(* Schneider Machine Expert - Basic project Zımpara-DIGITALINOUT, file version 1.8.0.0 *)
(* ProjectInformations: Name=Yeni proje *)

HARDWARE
  Cpu 0: TM221ME16T/G
  ModuleExtensionObject 0: TM3DI8/G
  ModuleExtensionObject 1: TM3AQ2/G
  EthernetConfiguration: NetworkName=M221, IpAllocationMode=FixedAddress, IpAddress=192.168.0.15, SubnetMask=255.255.255.0
  SerialLineConfiguration: Baud=Baud19200, Parity=ParityNone, DataBits=DataBits8, StopBits=StopBits1, PhysicalMedium=PhysicalMediumRs485, TransmissionMode=TransmissionModeModbusRtu, SlaveId=1, Addressing=SlaveAddressing
  MastTask: UsePeriodScanMode=false, PeriodScan=100
  FastTask: Period=255
  CpuBehavior: StartingMode=StartAsPreviousState, AutoSaveRamOnEeprom=true, WatchdogPeriod=250

SYMBOLS  (address, symbol, comment, settings)
  %M0         "HMI/OSILASYON YUKARI"
  %M1         "HMI/OSILASYON AŞAĞI"
  %M2         "HMI/FIRÇA  YUKARI"
  %M3         "HMI/FIRÇA  AŞAĞI"
  %M4         "HMI BANT START"
  %M5         "HMI OSILASYON START"
  %M6         "427/FIRCA INVERTOR"
  %M7         "428/VALF"
  %M8         "STOP"
  %M9         "HAFIZADAN ENCODERLERI ÇEK"
  %M10        "ENC 1 PRESET/OSILASYON ENC"
  %M11        "ENC 2 PRESET/FIRÇA ENC"
  %M12        "ENC_1_SIFIRLAMA/OSILASYON ENC"
  %M13        "ENC_2_SIFIRLAMA/FIRÇA ENC"
  %M16        "ENCODER2 ÇIKIŞ1"
  %M17        "ENCODER2 ÇIKIŞ2"
  %M18        "ENCODER2 ÇIKIŞ3"
  %M19        "ENCODER2 ÇIKIŞ4"
  %M21        "ENCODER 2 ÇIKIŞ1"
  %M22        "ENCODER 2 ÇIKIŞ2"
  %M23        "ENCODER 2 ÇIKIŞ3"
  %M24        "ENCODER 2 ÇIKIŞ4"
  %M26        "OSILASYON YÜKSEKLİK AYAR"
  %M27        "OSİLASYON YUKARI SET"
  %M28        "OSİLASYON AŞAĞI SET"
  %M29        "FIRÇA_YÜKSEKLİK_AYAR"
  %M30        "FIRÇA_YUKARI_SET"
  %M31        "FIRÇA_AŞAĞI_SET"
  %M32        "SQ5 CEVAP1"
  %M33        "SQ5 CEVAP2"
  %M201       "OSILASYON_KALIBRASYON"
  %S93      SB_MWBACKUP  "User set this bit to 1 to store the %MW variable in the flash (up to 2000)"
  %S94      SB_MWRESTORE  "User set this bit to 1 to restore the saved data"
  %SW148    SW_NBPERS  "Number of persistent variables (maximum 2000)"
  %MW1        "ENCODER 1 ÖN AYAR"
  %MW2        "ENCODER 2 ÖN AYAR"
  %MW30       "OSİLASYON SÜRÜCÜSÜ ANALOG ÇIKIŞ"
  %MW34       "ARKA FIRÇA SÜRÜCÜSÜ ANALOG ÇIKIŞ"
  %MW50       "BİRİNCİ ENKODER ANLIK DEĞERİ"
  %MW52       "İKİNCİ ENKODER ANLIK  DEĞERİ"
  %MF21       "2.ENCODER FLOAT DEĞERİ(MM)"
  %MF23       "1.ENKODER FLOAT DEĞERİ(MM)"
  %MF60       "ENC 1 FLOAT"
  %MF64       "OSILASYON MM YUKSEKLIK"
  %MF68       "OSILASYON ISTENEN YUKSEKLIK"
  %MF72       "ENC 2 FLOAT DEĞER"
  %MF76       "FIRÇA MM YÜKSEKLIK"
  %MF80       "FIRÇA ISTENEN YÜKSEKLIK"
  %MF84       "ENCODER 1 ÖN AYAR MM"
  %MF88       "ENCODER 1 ÖN AYAR INTEGER"
  %C0         "HAFIZADAN ENKODERLERİ ÇEK"
  %R0         "ENKODER 1 HAFIZAYA AT"
  %R1         "ENKODER 2 HAFIZAYA AT"
  %I0.0       "403/FIRÇA1 ÜST SINIR ANAHTARI"
  %I0.1       "402/FIRÇA1 ALT SINIR ANAHTARI"
  %I0.2       "405/FIRÇA2/ÜST SINIR ANAHTARI"
  %I0.3       "404/FIRÇA2/ ALT SINIR ANAHTARI"
  %I0.4       "SQ5(ÖN ARKA MESAFE SWITCHI)"
  %Q0.0       "421/OSİLASYON YUKARI"
  %Q0.1       "422/OSİLASYON AŞAĞI"
  %Q0.2       "423/FIRÇA 2 YUKARI"
  %Q0.3       "424/FIRÇA 2 AŞAĞI"
  %Q0.4       "425/BANT START"
  %Q0.5       "426/OSILASYON START"
  %Q0.6       "427/FIRCA INVERTER"
  %Q0.7       "428/VALF"
  %HSC0       "FIRÇA1/ENKODER"  [Type=CounterOrDownCounterBiPhasesX1, Preset=0, DedicatedInputs(DedicatedInput(Activated=true), DedicatedInput(Activated=true)), ReflexOutputs(ReflexOutput(Activated=false, LessThanS0=false, GreaterOrEqualThanS0=false, GreaterOrEqualThanS1=false), ReflexOutput(Activated=false, LessThanS0=false, GreaterOrEqualThanS0=false, GreaterOrEqualThanS1=false)), Thresholds(Threshold(ThresholdType=NotUsed, Pri]
  %HSC1       "FIRÇA2/ENKODER"  [Type=CounterOrDownCounterBiPhasesX1, Preset=0, DedicatedInputs(DedicatedInput(Activated=true), DedicatedInput(Activated=true)), ReflexOutputs(ReflexOutput(Activated=false, LessThanS0=false, GreaterOrEqualThanS0=false, GreaterOrEqualThanS1=false), ReflexOutput(Activated=false, LessThanS0=false, GreaterOrEqualThanS0=false, GreaterOrEqualThanS1=false)), Thresholds(Threshold(ThresholdType=NotUsed, Pri]
  %I1.0       "403/FIRÇA UST SINIR SWITCH"
  %I1.1       "402/FIRÇA ALT SINIR SWITCH"
  %I1.2       "405/FIRÇA2/ÜST SINIR SWITCH"
  %I1.3       "404/FIRÇA2/ALT SINIR SWITCH"
  %QW2.0      [Type=Type_0_10V, Scope=Scope_Customized, Minimum=0, Maximum=100]
  %QW2.1      [Type=Type_0_10V, Scope=Scope_Customized, Minimum=0, Maximum=100]

POU Yeni POU
  (* SectionNumber=1 *)

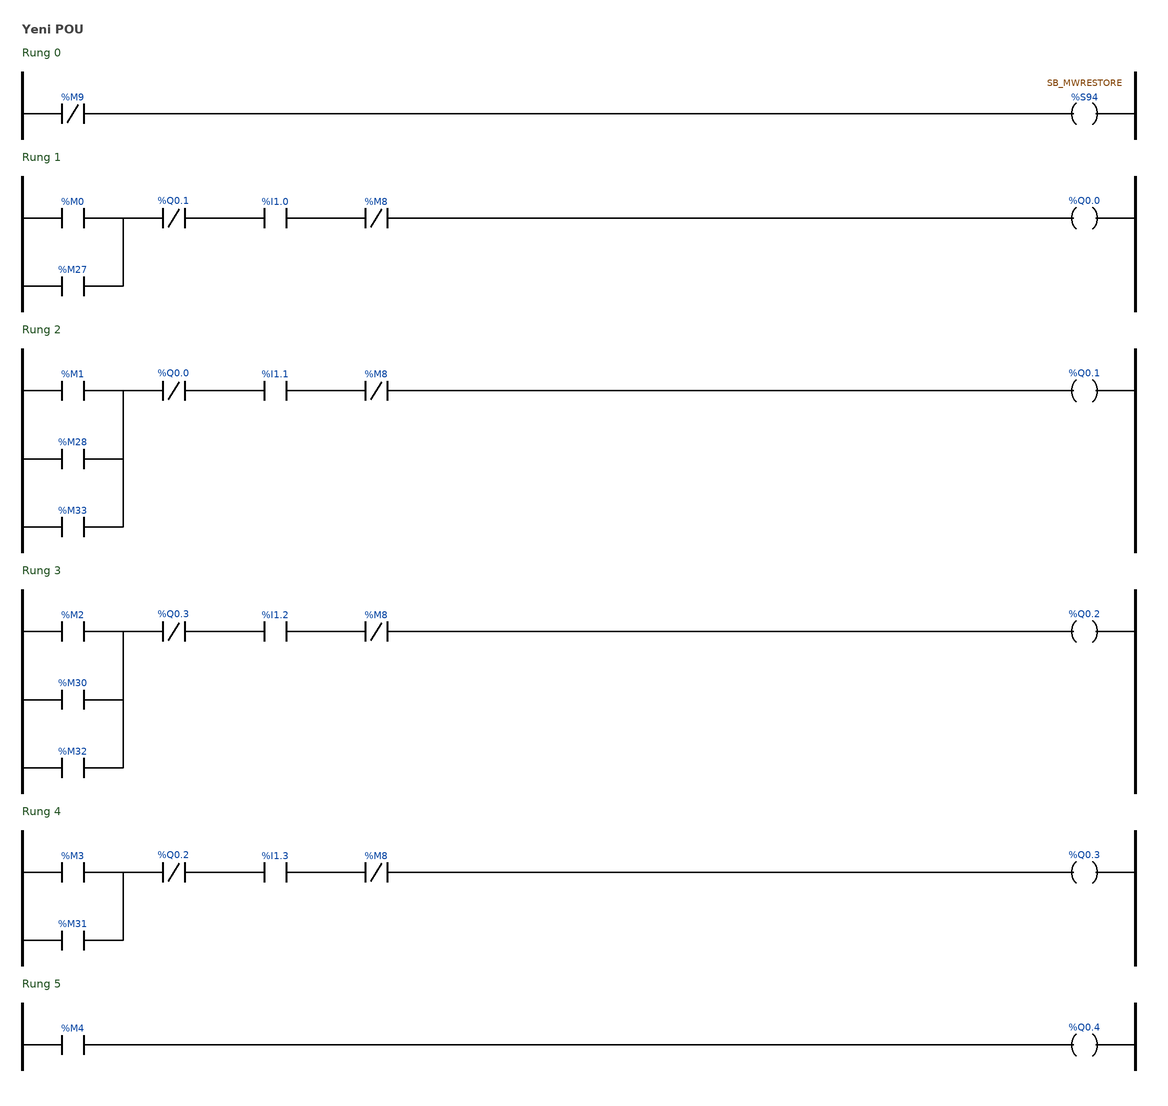

// Rung 0
  LDN %M9
  ST %S94                 (* SB_MWRESTORE *)
  // as ST:
  //   SB_MWRESTORE := NOT %M9;

// Rung 1
  LD %M0
  OR %M27
  ANDN %Q0.1
  AND %I1.0
  ANDN %M8
  ST %Q0.0
  // as ST:
  //   %Q0.0 := (%M0 OR %M27) AND NOT %Q0.1 AND %I1.0 AND NOT %M8;

// Rung 2
  LD %M1
  OR %M28
  OR %M33
  ANDN %Q0.0
  AND %I1.1
  ANDN %M8
  ST %Q0.1
  // as ST:
  //   %Q0.1 := (%M1 OR %M28 OR %M33) AND NOT %Q0.0 AND %I1.1 AND NOT %M8;

// Rung 3
  LD %M2
  OR %M30
  OR %M32
  ANDN %Q0.3
  AND %I1.2
  ANDN %M8
  ST %Q0.2
  // as ST:
  //   %Q0.2 := (%M2 OR %M30 OR %M32) AND NOT %Q0.3 AND %I1.2 AND NOT %M8;

// Rung 4
  LD %M3
  OR %M31
  ANDN %Q0.2
  AND %I1.3
  ANDN %M8
  ST %Q0.3
  // as ST:
  //   %Q0.3 := (%M3 OR %M31) AND NOT %Q0.2 AND %I1.3 AND NOT %M8;

// Rung 5
  LD %M4
  ST %Q0.4
  // as ST:
  //   %Q0.4 := %M4;

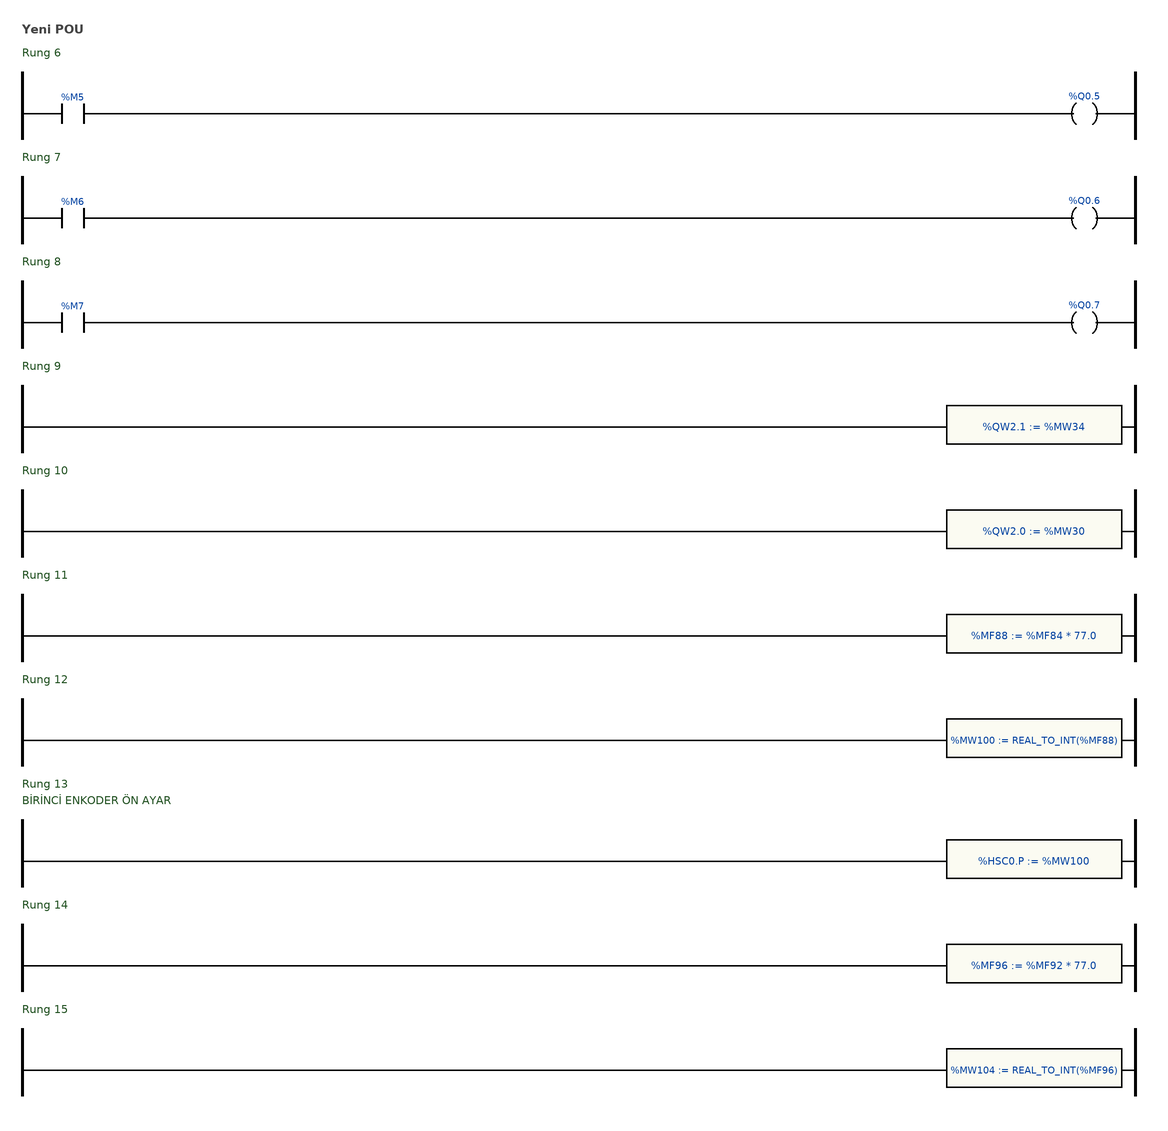

// Rung 6
  LD %M5
  ST %Q0.5
  // as ST:
  //   %Q0.5 := %M5;

// Rung 7
  LD %M6
  ST %Q0.6
  // as ST:
  //   %Q0.6 := %M6;

// Rung 8
  LD %M7
  ST %Q0.7
  // as ST:
  //   %Q0.7 := %M7;

// Rung 9
  LD 1
  [ %QW2.1 := %MW34 ]
  // as ST:
  //   %QW2.1 := %MW34;

// Rung 10
  LD 1
  [ %QW2.0 := %MW30 ]
  // as ST:
  //   %QW2.0 := %MW30;

// Rung 11
  LD 1
  [ %MF88 := %MF84 * 77.0 ]
  // as ST:
  //   %MF88 := %MF84  *  77.0;

// Rung 12
  LD 1
  [ %MW100 := REAL_TO_INT ( %MF88 ) ]
  // as ST:
  //   %MW100 := REAL_TO_INT ( %MF88 );

// Rung 13
// BİRİNCİ ENKODER ÖN AYAR
  LD 1
  [ %HSC0.P := %MW100 ]
  // as ST:
  //   %HSC0.P := %MW100;

// Rung 14
  LD 1
  [ %MF96 := %MF92 * 77.0 ]
  // as ST:
  //   %MF96 := %MF92  *  77.0;

// Rung 15
  LD 1
  [ %MW104 := REAL_TO_INT ( %MF96 ) ]
  // as ST:
  //   %MW104 := REAL_TO_INT ( %MF96 );

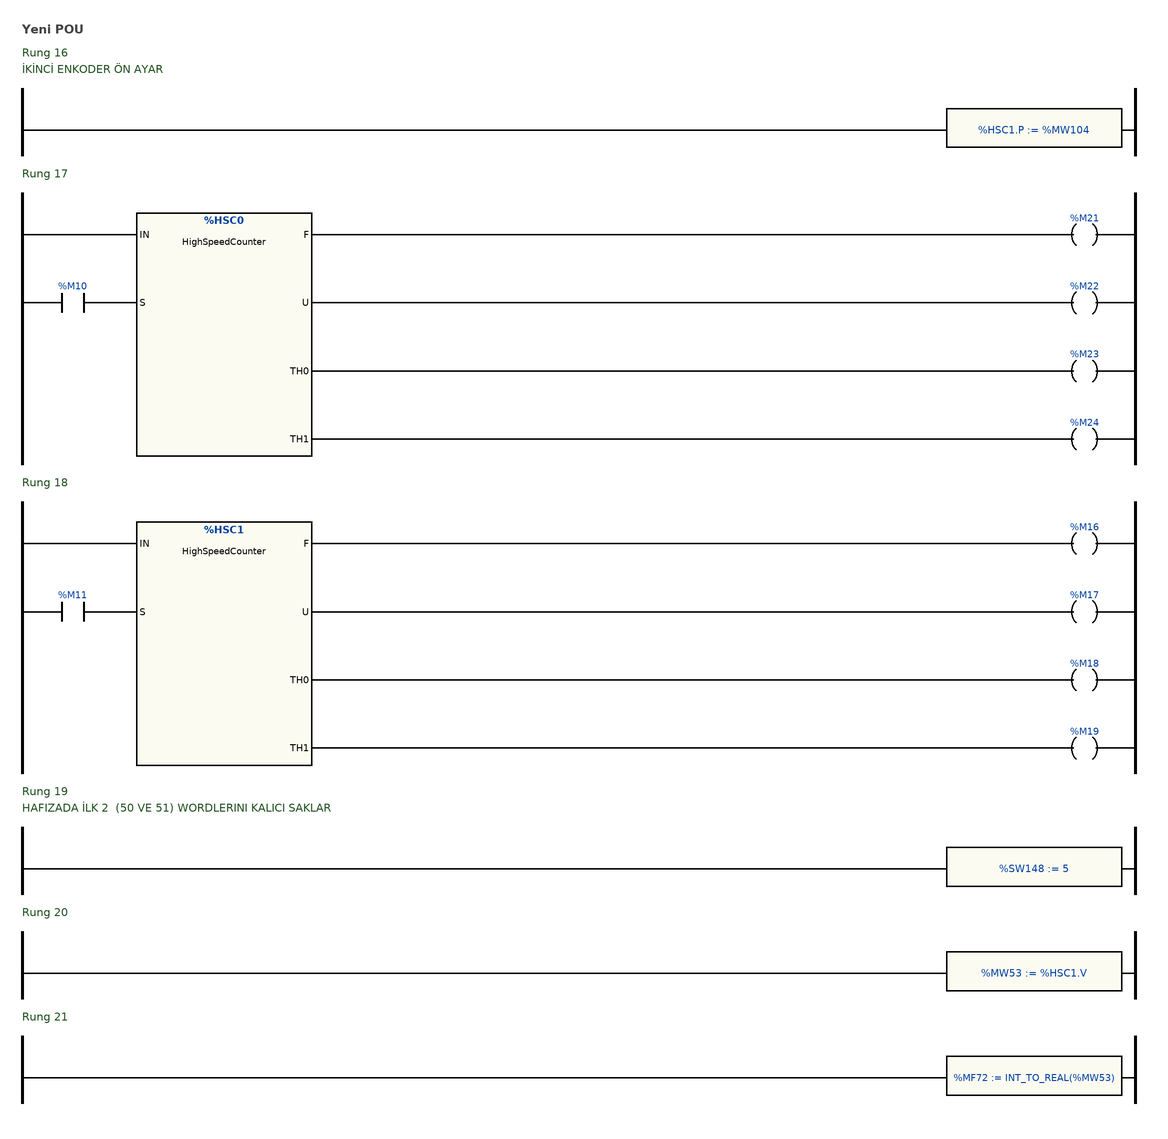

// Rung 16
// İKİNCİ ENKODER ÖN AYAR
  LD 1
  [ %HSC1.P := %MW104 ]
  // as ST:
  //   %HSC1.P := %MW104;

// Rung 17
  BLK %HSC0
  LD 1
  IN
  LD %M10
  S
  OUT_BLK
  LD F
  ST %M21
  LD U
  ST %M22
  LD TH0
  ST %M23
  LD TH1
  ST %M24
  END_BLK
  // as ST:
  //   %HSC0(IN := TRUE, S := %M10);
  //   %M21 := %HSC0.F;
  //   %M22 := %HSC0.U;
  //   %M23 := %HSC0.TH0;
  //   %M24 := %HSC0.TH1;

// Rung 18
  BLK %HSC1
  LD 1
  IN
  LD %M11
  S
  OUT_BLK
  LD F
  ST %M16
  LD U
  ST %M17
  LD TH0
  ST %M18
  LD TH1
  ST %M19
  END_BLK
  // as ST:
  //   %HSC1(IN := TRUE, S := %M11);
  //   %M16 := %HSC1.F;
  //   %M17 := %HSC1.U;
  //   %M18 := %HSC1.TH0;
  //   %M19 := %HSC1.TH1;

// Rung 19
// HAFIZADA İLK 2  (50 VE 51) WORDLERINI KALICI SAKLAR
  LD 1
  [ %SW148 := 5 ]         (* SW_NBPERS *)
  // as ST:
  //   SW_NBPERS := 5;

// Rung 20
  LD 1
  [ %MW53 := %HSC1.V ]
  // as ST:
  //   %MW53 := %HSC1.V;

// Rung 21
  LD 1
  [ %MF72 := INT_TO_REAL ( %MW53 ) ]
  // as ST:
  //   %MF72 := INT_TO_REAL ( %MW53 );

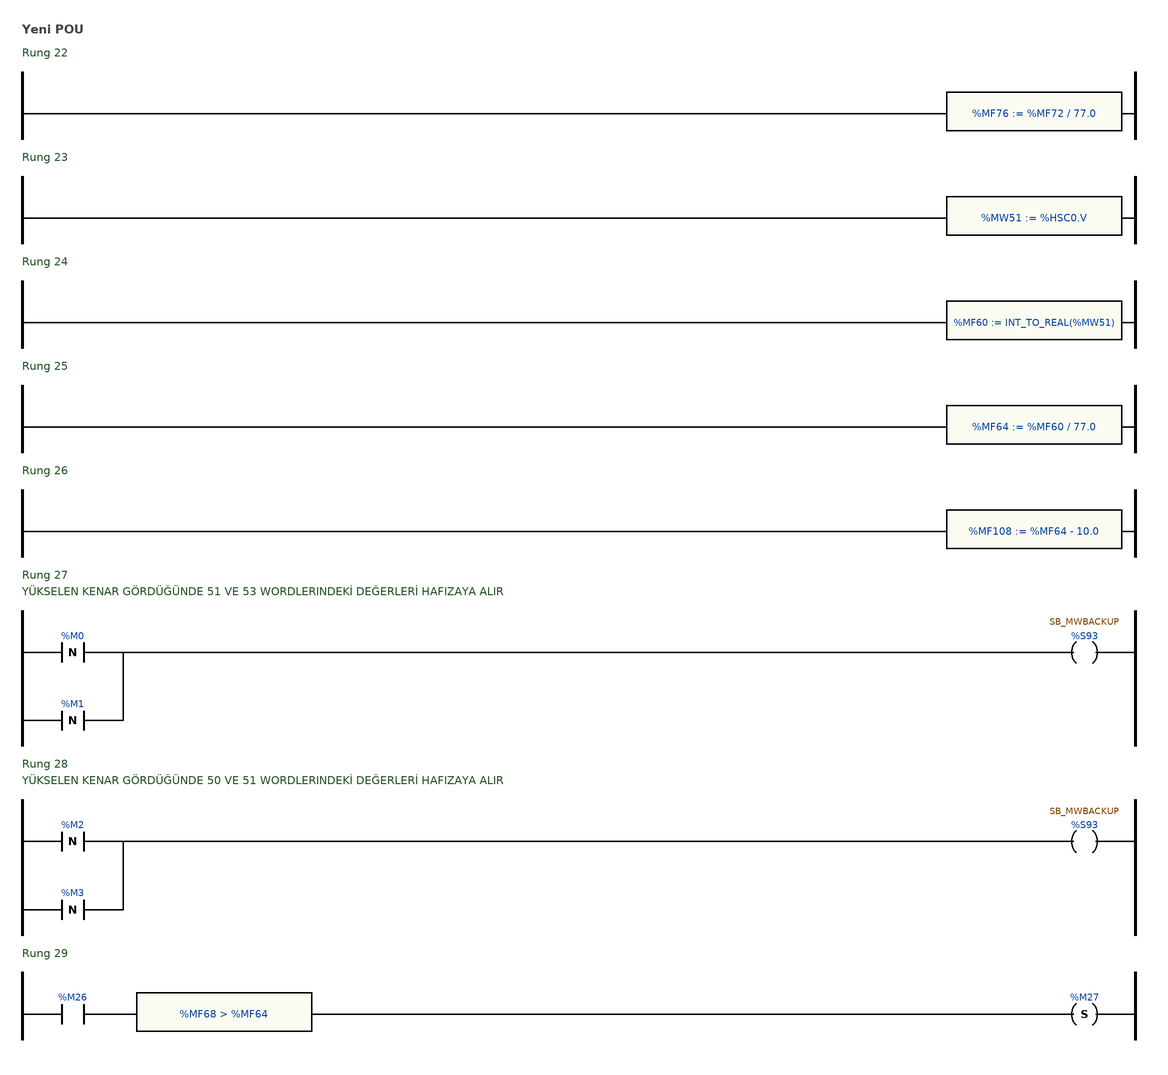

// Rung 22
  LD 1
  [ %MF76 := %MF72 / 77.0 ]
  // as ST:
  //   %MF76 := %MF72  /  77.0;

// Rung 23
  LD 1
  [ %MW51 := %HSC0.V ]
  // as ST:
  //   %MW51 := %HSC0.V;

// Rung 24
  LD 1
  [ %MF60 := INT_TO_REAL ( %MW51 ) ]
  // as ST:
  //   %MF60 := INT_TO_REAL ( %MW51 );

// Rung 25
  LD 1
  [ %MF64 := %MF60 / 77.0 ]
  // as ST:
  //   %MF64 := %MF60  /  77.0;

// Rung 26
  LD 1
  [ %MF108 := %MF64 - 10.0 ]
  // as ST:
  //   %MF108 := %MF64  -  10.0;

// Rung 27
// YÜKSELEN KENAR GÖRDÜĞÜNDE 51 VE 53 WORDLERINDEKİ DEĞERLERİ HAFIZAYA ALIR
  LDF %M0
  ORF %M1
  ST %S93                 (* SB_MWBACKUP *)
  // as ST:
  //   SB_MWBACKUP := FALLING(%M0) OR FALLING(%M1);

// Rung 28
// YÜKSELEN KENAR GÖRDÜĞÜNDE 50 VE 51 WORDLERINDEKİ DEĞERLERİ HAFIZAYA ALIR
  LDF %M2
  ORF %M3
  ST %S93                 (* SB_MWBACKUP *)
  // as ST:
  //   SB_MWBACKUP := FALLING(%M2) OR FALLING(%M3);

// Rung 29
  LD %M26
  AND [ %MF68 > %MF64 ]
  S %M27
  // as ST:
  //   IF %M26 AND %MF68 > %MF64 THEN %M27 := TRUE; END_IF;

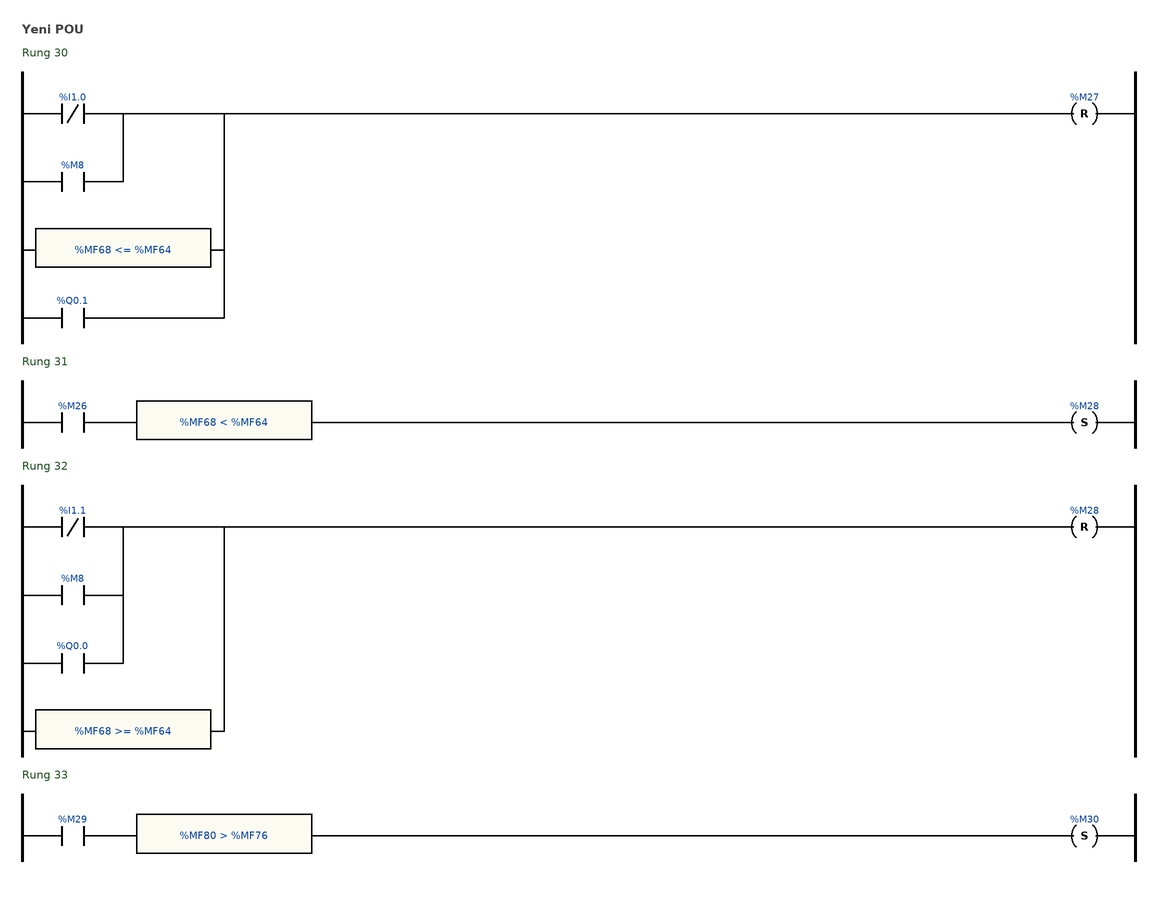

// Rung 30
  LDN %I1.0
  OR %M8
  OR [ %MF68 <= %MF64 ]
  OR %Q0.1
  R %M27
  // as ST:
  //   IF NOT %I1.0 OR %M8 OR %MF68 <= %MF64 OR %Q0.1 THEN %M27 := FALSE; END_IF;

// Rung 31
  LD %M26
  AND [ %MF68 < %MF64 ]
  S %M28
  // as ST:
  //   IF %M26 AND %MF68 < %MF64 THEN %M28 := TRUE; END_IF;

// Rung 32
  LDN %I1.1
  OR %M8
  OR %Q0.0
  OR [ %MF68 >= %MF64 ]
  R %M28
  // as ST:
  //   IF NOT %I1.1 OR %M8 OR %Q0.0 OR %MF68 >= %MF64 THEN %M28 := FALSE; END_IF;

// Rung 33
  LD %M29
  AND [ %MF80 > %MF76 ]
  S %M30
  // as ST:
  //   IF %M29 AND %MF80 > %MF76 THEN %M30 := TRUE; END_IF;

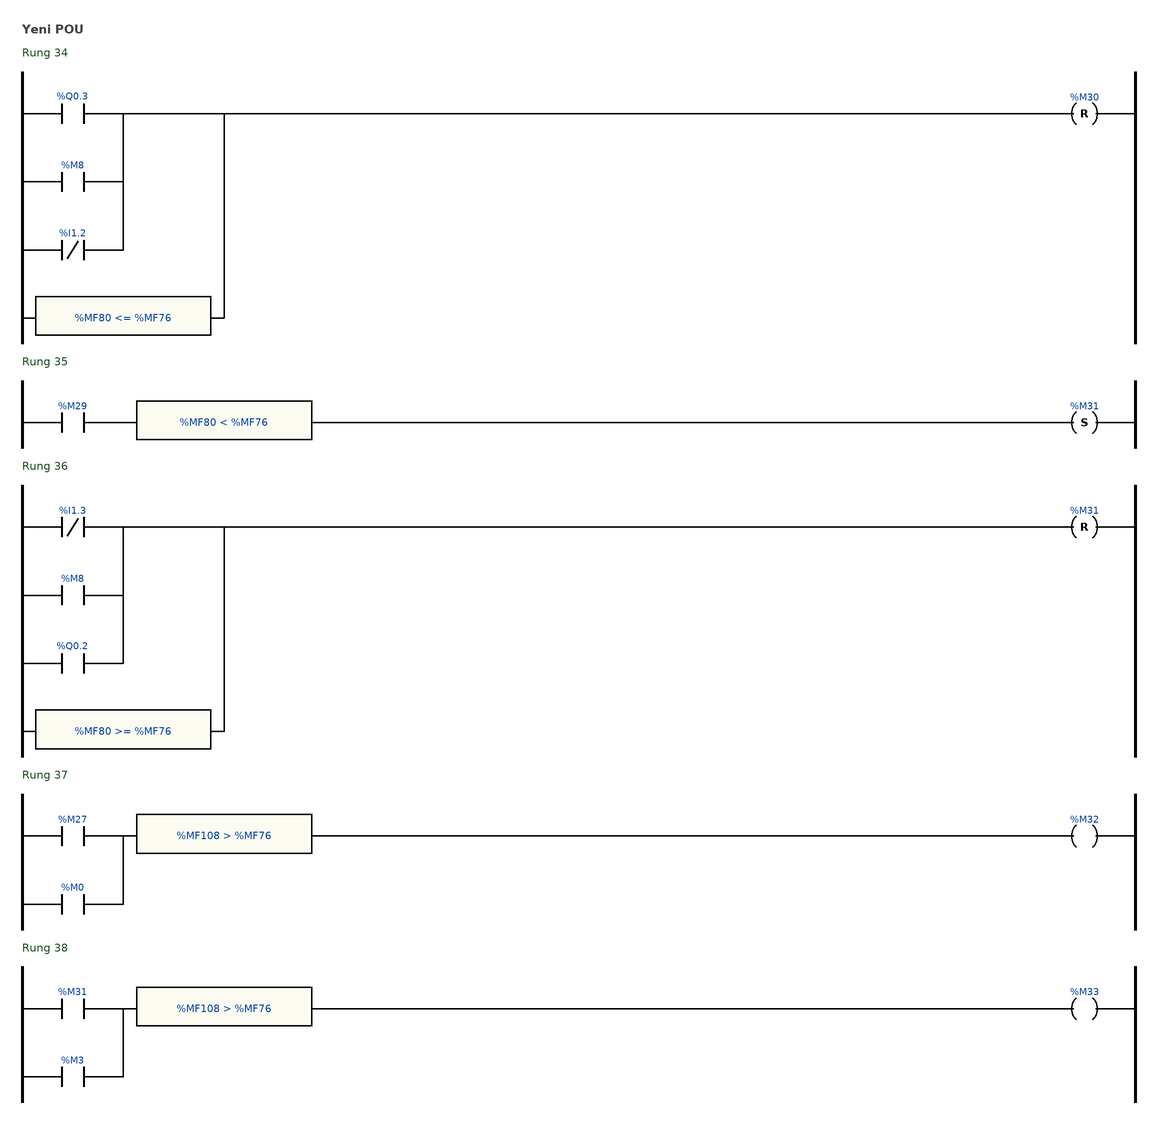

// Rung 34
  LD %Q0.3
  OR %M8
  ORN %I1.2
  OR [ %MF80 <= %MF76 ]
  R %M30
  // as ST:
  //   IF %Q0.3 OR %M8 OR NOT %I1.2 OR %MF80 <= %MF76 THEN %M30 := FALSE; END_IF;

// Rung 35
  LD %M29
  AND [ %MF80 < %MF76 ]
  S %M31
  // as ST:
  //   IF %M29 AND %MF80 < %MF76 THEN %M31 := TRUE; END_IF;

// Rung 36
  LDN %I1.3
  OR %M8
  OR %Q0.2
  OR [ %MF80 >= %MF76 ]
  R %M31
  // as ST:
  //   IF NOT %I1.3 OR %M8 OR %Q0.2 OR %MF80 >= %MF76 THEN %M31 := FALSE; END_IF;

// Rung 37
  LD %M27
  OR %M0
  AND [ %MF108 > %MF76 ]
  ST %M32
  // as ST:
  //   %M32 := (%M27 OR %M0) AND %MF108 > %MF76;

// Rung 38
  LD %M31
  OR %M3
  AND [ %MF108 > %MF76 ]
  ST %M33
  // as ST:
  //   %M33 := (%M31 OR %M3) AND %MF108 > %MF76;

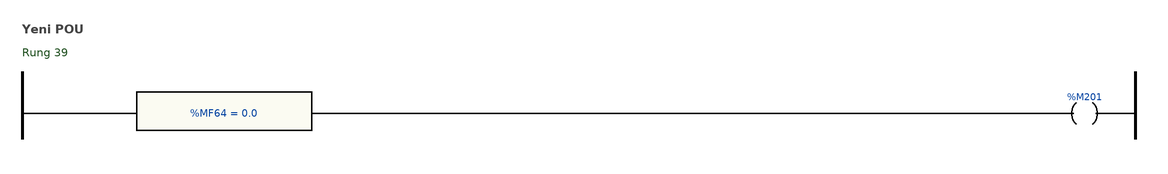

// Rung 39
  LD 1
  AND [ %MF64 = 0.0 ]
  ST %M201
  // as ST:
  //   %M201 := %MF64 = 0.0;
